Staubli VAL3: increase.pgx

public program increase(num x_nType)
begin
  // increase the size plus 1
  switch x_nType
    case 0
      // START LIST
      saveCycle:nDoneStart[cycleStatus:nProg]=saveCycle:nDoneStart[cycleStatus:nProg]+1
    break
    case 1
      // PROCESS LIST
      saveCycle:nDoneCycle[0]=saveCycle:nDoneCycle[0]+1
    break
    case 2
      // END LIST
      saveCycle:nDoneEnd[cycleStatus:nProg]=saveCycle:nDoneEnd[cycleStatus:nProg]+1
    break
  endSwitch
end
